FUNCTION_BLOCK FutureMCStopCreator IMPLEMENTS I_TaskCreator
VAR_INPUT
END_VAR
VAR_OUTPUT
END_VAR
VAR
	_axis: REFERENCE TO AXIS_REF;
	_deceleration: MC_LREAL;
	_jerk		: MC_LREAL;
	_option : ST_MoveOptions;
	_buffer_mode : MC_BufferMode;
END_VAR

{warning 'add method implementation '}
METHOD create_future : I_Future
VAR_INPUT
	(* Specify future name*)
	future_name	: STRING;
END_VAR
VAR
	_p_future : POINTER TO FutureMCStop;
END_VAR
_p_future := __NEW(FutureMCStop);
_p_future^.future_name := future_name;
_p_future^.set_parameters(_axis, _deceleration, _jerk);
_p_future^.set_options(_option);
create_future := _p_future^;
END_METHOD

{warning 'add method implementation '}
METHOD destroy_future : I_Future
VAR_INPUT
	(* Specify future instance whtat you want to delete.*)
	future	: I_Future;
END_VAR
VAR
	_p_future : POINTER TO FutureMCStop;
END_VAR
IF __QUERYPOINTER(future, _p_future) THEN
	__DELETE(_p_future);
	IF _p_future = 0  THEN
		destroy_future := 0;
	END_IF
END_IF
END_METHOD

METHOD set_options : BOOL
VAR_INPUT
	option : ST_MoveOptions;
END_VAR
_option := option;
END_METHOD

METHOD set_parameters : BOOL
VAR_INPUT
	axis : REFERENCE TO AXIS_REF;
	deceleration	: MC_LREAL;		// Set deceleration in case let moving axis halt.
	jerk			: MC_LREAL;		// Set jerk in case let moving axis halt.
END_VAR
_axis REF= axis;
_deceleration := deceleration;
_jerk := jerk;
END_METHOD

END_FUNCTION_BLOCK

(* stored: Version 1.1.0.1, ProductVersion 3.1.4026.17
   POU FutureMCStopCreator: Id {2aa0840a-ea83-4839-96a4-e982629c2128}, SpecialFunc None
   Method create_future: Id {cde46ba2-2def-45b1-8a5c-0125d157852f}
   Method destroy_future: Id {701772d1-8e6f-4e4f-9c7c-933fa6c3ea4e}
   Method set_options: Id {ca47d14d-5f66-4c9c-a4cc-9949f1d4f8de}
   Method set_parameters: Id {02982528-c91a-4c66-b968-8b28ea9a4815} *)
